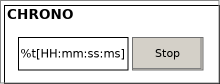
VISUALIZATION CHRONO  // 220x84
VAR_IN_OUT
	m_input_CHRONO : TON;
END_VAR
    Rectangle (4,5 216x79), "CHRONO"
    RoundedRectangle (18,37 110x33), "%t[HH:mm:ss:ms]", text variable: m_input_CHRONO.ET
        OnMouseDown: write the text variable via VisuDialogs.Numpad, min 7, max 10
    Button (132,37 71x33), "Start", invisible if: m_input_CHRONO.IN
        OnMouseClick: execute { m_input_CHRONO.IN := TRUE; }
    Button (132,37 71x33), "Stop", invisible if: NOT m_input_CHRONO.IN
        OnMouseClick: execute { m_input_CHRONO.IN := FALSE; }
END_VISUALIZATION

(* stored: Version 1.1.0.1, ProductVersion 3.1.4024.10
   Visu CHRONO: Id {254bdfb3-42b0-47da-8f2d-7ef975198274} *)
